FUNCTION_BLOCK FB_Hoval EXTENDS FbModbusTcpBase
// 07.05.2025 Elmar Vögel
VAR_INPUT
  END_VAR
VAR_OUTPUT
  HalleMattenrain11Soll       : LREAL;
  HalleMattenrain11VLIst      : LREAL;
  RadGravierraumSoll          : LREAL;
  FbhGaderobeWCSoll           : LREAL;
  RadGravierraumIst           : LREAL;
  FbhGaderobeWCIst            : LREAL;
  LufterhitzerLagerSoll       : LREAL;
  BueroHusSoll                : LREAL;
  LufterhitzerLagerIst        : LREAL;
  BueroHusIst                 : LREAL;
  HalleMattenrain11Strategie  : INT;
  RadGravierraumStrategie     : INT;
  FbhGaderobeWCStrategie      : INT;
  LufterhitzerLagerStrategie  : INT;
  BueroHusStrategie           : INT;
END_VAR

VAR CONSTANT
  cDelaySend : TIME:= T#1S;  
END_VAR

VAR
  iState      : INT;
  mPoll       : TON:= (PT:= T#1S);

  mReg        : ARRAY[0..10] OF WORD;
END_VAR

{region "Basis"}
  SUPER^();
{endregion}
{region "Modbus bearbeiten"}
  CASE iState OF
  0:  

    mPoll(IN:= TRUE);
    IF mPoll.Q THEN

      mPoll(IN:= FALSE);
  
      mCmd.UnitID   := 16#3;
      mCmd.Funktion := ModbusFunktion.ReadRegs;
      mCmd.MBAddr   := 16#06DC; // 1756
      mCmd.Quantity := 1; 
      mCmd.DatenAddr:= ADR(mReg);
      mCmd.DatenLen := SIZEOF(mReg);
  
      iState:= 100;
    END_IF

  100: SendNext(iState + 1);
  101:
    IF Empfang(cDelaySend) THEN

      IF NOT Error THEN
        HalleMattenrain11Soll:= TO_LREAL(mReg[0]) / 10.0;
      END_IF
         
      mCmd.UnitID   := 16#3;
      mCmd.Funktion := ModbusFunktion.ReadRegs;
      mCmd.MBAddr   := 16#06F3; // 1779
      mCmd.Quantity := 1; 
      mCmd.DatenAddr:= ADR(mReg);
      mCmd.DatenLen := SIZEOF(mReg);

      iState:= 110; 
    END_IF

  110: SendNext(iState + 1);
  111:
    IF Empfang(cDelaySend) THEN

      IF NOT Error THEN
        HalleMattenrain11VLIst:= TO_LREAL(mReg[0]) / 10.0;
      END_IF
         
      mCmd.UnitID   := 16#9;
      mCmd.Funktion := ModbusFunktion.ReadRegs;
      mCmd.MBAddr   := 16#1179; // 4473
      mCmd.Quantity := 2; 
      mCmd.DatenAddr:= ADR(mReg);
      mCmd.DatenLen := SIZEOF(mReg);

      iState:= 120; 
    END_IF

  120: SendNext(iState + 1);
  121:
    IF Empfang(cDelaySend) THEN

      IF NOT Error THEN
        RadGravierraumSoll:= TO_LREAL(mReg[0]) / 10.0;
        FbhGaderobeWCSoll := TO_LREAL(mReg[1]) / 10.0;
      END_IF
         
      mCmd.UnitID   := 16#9;
      mCmd.Funktion := ModbusFunktion.ReadRegs;
      mCmd.MBAddr   := 16#118A; // 4490
      mCmd.Quantity := 2; 
      mCmd.DatenAddr:= ADR(mReg);
      mCmd.DatenLen := SIZEOF(mReg);

      iState:= 130; 
    END_IF

  130: SendNext(iState + 1);
  131:
    IF Empfang(cDelaySend) THEN

      IF NOT Error THEN
        RadGravierraumIst:= TO_LREAL(mReg[0]) / 10.0;
        FbhGaderobeWCIst := TO_LREAL(mReg[1]) / 10.0;
      END_IF
         
      mCmd.UnitID   := 16#A;
      mCmd.Funktion := ModbusFunktion.ReadRegs;
      mCmd.MBAddr   := 16#11D7; // 4567
      mCmd.Quantity := 2; 
      mCmd.DatenAddr:= ADR(mReg);
      mCmd.DatenLen := SIZEOF(mReg);

      iState:= 140; 
    END_IF

  140: SendNext(iState + 1);
  141:
    IF Empfang(cDelaySend) THEN

      IF NOT Error THEN
        LufterhitzerLagerSoll:= TO_LREAL(mReg[0]) / 10.0;
        BueroHusSoll         := TO_LREAL(mReg[1]) / 10.0;
      END_IF
         
      mCmd.UnitID   := 16#A;
      mCmd.Funktion := ModbusFunktion.ReadRegs;
      mCmd.MBAddr   := 16#11E8; // 4584
      mCmd.Quantity := 2; 
      mCmd.DatenAddr:= ADR(mReg);
      mCmd.DatenLen := SIZEOF(mReg);

      iState:= 150; 
    END_IF

  150: SendNext(iState + 1);
  151:
    IF Empfang(cDelaySend) THEN

      IF NOT Error THEN
        LufterhitzerLagerIst:= TO_LREAL(mReg[0]) / 10.0;
        BueroHusIst         := TO_LREAL(mReg[1]) / 10.0;
      END_IF
         
      mCmd.UnitID   := 16#3;
      mCmd.Funktion := ModbusFunktion.ReadRegs;
      mCmd.MBAddr   := 16#6C02; // 27650
      mCmd.Quantity := 1; 
      mCmd.DatenAddr:= ADR(mReg);
      mCmd.DatenLen := SIZEOF(mReg);

      iState:= 160; 
    END_IF

  160: SendNext(iState + 1);
  161:
    IF Empfang(cDelaySend) THEN

      IF NOT Error THEN
        HalleMattenrain11Strategie:= TO_INT(mReg[0]);
      END_IF
         
      mCmd.UnitID   := 16#9;
      mCmd.Funktion := ModbusFunktion.ReadRegs;
      mCmd.MBAddr   := 16#78BB; // 30907
      mCmd.Quantity := 2; 
      mCmd.DatenAddr:= ADR(mReg);
      mCmd.DatenLen := SIZEOF(mReg);

      iState:= 170; 
    END_IF

  170: SendNext(iState + 1);
  171:
    IF Empfang(cDelaySend) THEN

      IF NOT Error THEN
        RadGravierraumStrategie:= TO_INT(mReg[0]);
        FbhGaderobeWCStrategie := TO_INT(mReg[1]);
      END_IF
         
      mCmd.UnitID   := 16#A;
      mCmd.Funktion := ModbusFunktion.ReadRegs;
      mCmd.MBAddr   := 16#78BE; // 30910
      mCmd.Quantity := 2; 
      mCmd.DatenAddr:= ADR(mReg);
      mCmd.DatenLen := SIZEOF(mReg);

      iState:= 180; 
    END_IF

  180: SendNext(iState + 1);
  181:
    IF Empfang(cDelaySend) THEN

      IF NOT Error THEN
        LufterhitzerLagerStrategie:= TO_INT(mReg[0]);
        BueroHusStrategie         := TO_INT(mReg[1]);
      END_IF
         
      iState:= 800; 
    END_IF

  800:
    // Fertig
    iState:= 0;
  END_CASE
{endregion}

METHOD PRIVATE SendNext : BOOL
VAR_INPUT
  StepNext : INT;
END_VAR

  SendNext:= FALSE;
  IF SUPER^.Send() THEN

    iState:= StepNext;
    SendNext:= TRUE;
  END_IF
END_METHOD

END_FUNCTION_BLOCK

(* stored: Version 1.1.0.1, ProductVersion 3.1.4024.15
   POU FB_Hoval: Id {81f9879f-29c7-470a-91d2-1d4240ff5b65}, SpecialFunc None
   Method SendNext: Id {3e1e2460-a785-4514-9c77-273926321810} *)
